(* Logix 5000 project; controller Transcat_L33ER vendor 1 type 14 code 107 rev 32.11; software revision 32.02; part 2 of 2 *)
(* tags used below, declared in another part *)
   alwaysOFF : BOOL;
   AnyAutoRun : BOOL;   // Bit that in on if ANY device is placed into Auto run (to signal pre-start beed)
   AnyManualRun : BOOL;   // Bit that in on if ANY device is placed into manual run (to signal pre-start beed)
   BeaconBlueLight : ALIAS FOR TC_Remote_IO:3:O.3;   // Blue Beacon Light
   BeaconGreenLight : ALIAS FOR TC_Remote_IO:3:O.2;   // Green Beacon Light
   BeaconRedLight : ALIAS FOR TC_Remote_IO:3:O.0;   // Red Beacon Light
   BeaconYellowLight : ALIAS FOR TC_Remote_IO:3:O.1;   // Yellow Beacon Light
   Beep : BOOL;   // Bit to Activte Beacon Alarm
   BeepNew : ALIAS FOR TC_Remote_IO:3:O.4;
   Device : Device[20];
   FT103 : BronkhorstFlowMeter;
   FT104 : BronkhorstFlowMeter;
   FT105 : BronkhorstFlowMeter;
   GF101 : Thayer_WB_Feeder;   // Thayer 1 Tags
   GF201 : Thayer_WB_Feeder;   // Thayer 2 Tags
   GF301 : Acrison_Feeder;   // GF103 - Small Feeder 1
   GreenFlashingOff : TIMER;
   GreenFlashingOn : TIMER;
   HMI_AllReset : BOOL;   // Bit to reset Auto/Man, AutoRun, RecipeRun, TimedRunEnable to 0 from HMI
   MSG_FROM_SLC500 : INT[10];
   MX101 : Howes_Mixer;
   MX201 : Howes_Mixer;
   StartBeepTimer : TIMER;   // Timer to sound the beep alarm before starting a device
   UpperHowesSpeed : INT;
   VF101 : Acrison_Feeder;   // Medium Feeder Tags
   VF201 : Acrison_Feeder;   // Small Feeder 2 Tags
   YellowFlashOff : TIMER;
   YellowFlashOn : TIMER;
   ZS101_RPM_Speed_UpperHowes : ALIAS FOR TC_Remote_IO:1:I.Ch3Data;   // Upper Howes Zero Speed Sensor RPM
   ZS102_RPM_Speed_LowerHowes : ALIAS FOR TC_Remote_IO:1:I.Ch4Data;   // Lower Howes Zero Speed Sensor RPM
(* MainProgram, continued *)

ROUTINE Light_Beacon   (* ladder *)
// Indicator Light Beacon
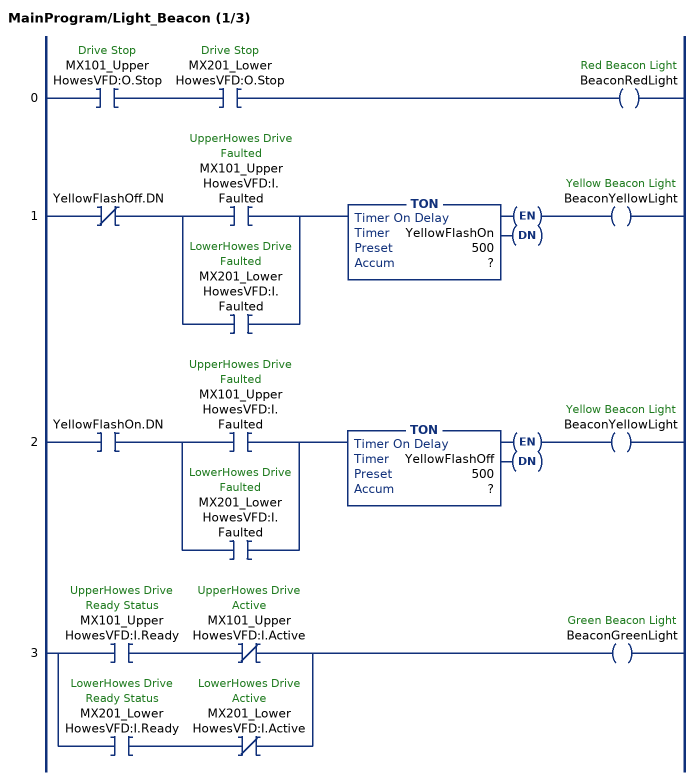
   0: XIC(MX101_UpperHowesVFD:O.Stop)XIC(MX201_LowerHowesVFD:O.Stop)OTE(BeaconRedLight);
   1: XIO(YellowFlashOff.DN)[XIC(MX101_UpperHowesVFD:I.Faulted) ,XIC(MX201_LowerHowesVFD:I.Faulted) ]TON(YellowFlashOn,?,?)OTE(BeaconYellowLight);
   2: XIC(YellowFlashOn.DN)[XIC(MX101_UpperHowesVFD:I.Faulted) ,XIC(MX201_LowerHowesVFD:I.Faulted) ]TON(YellowFlashOff,?,?)OTE(BeaconYellowLight);
   3: [XIC(MX101_UpperHowesVFD:I.Ready) XIO(MX101_UpperHowesVFD:I.Active) ,XIC(MX201_LowerHowesVFD:I.Ready) XIO(MX201_LowerHowesVFD:I.Active) ]OTE(BeaconGreenLight);
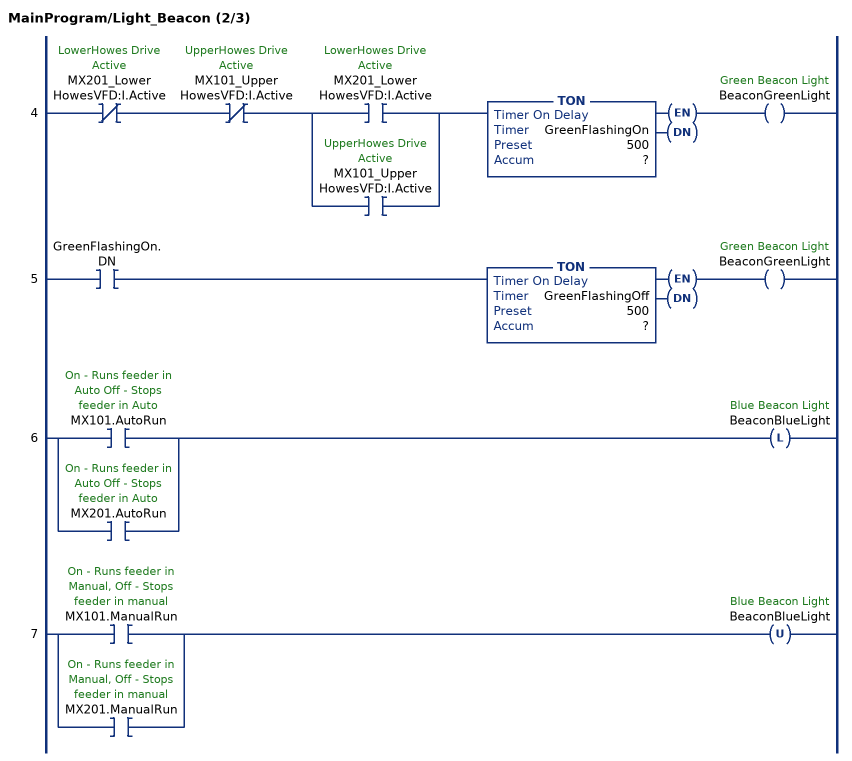
   4: XIO(MX201_LowerHowesVFD:I.Active)XIO(MX101_UpperHowesVFD:I.Active)[XIC(MX201_LowerHowesVFD:I.Active) ,XIC(MX101_UpperHowesVFD:I.Active) ]TON(GreenFlashingOn,?,?)OTE(BeaconGreenLight);
   5: XIC(GreenFlashingOn.DN)TON(GreenFlashingOff,?,?)OTE(BeaconGreenLight);
   6: [XIC(MX101.AutoRun) ,XIC(MX201.AutoRun) ]OTL(BeaconBlueLight);
   7: [XIC(MX101.ManualRun) ,XIC(MX201.ManualRun) ]OTU(BeaconBlueLight);
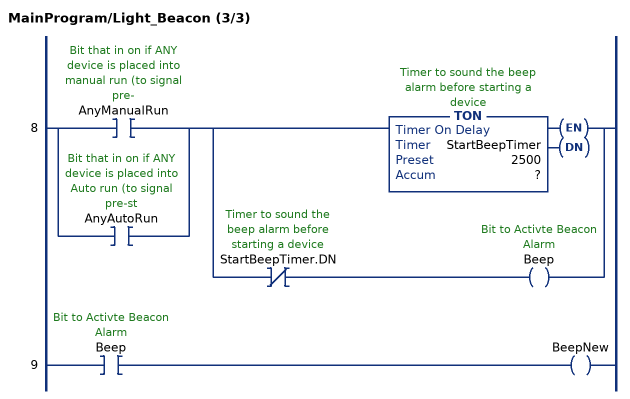
   8: [XIC(AnyManualRun) ,XIC(AnyAutoRun) ][TON(StartBeepTimer,?,?) ,XIO(StartBeepTimer.DN) OTE(Beep) ];
   9: XIC(Beep)OTE(BeepNew);
END_ROUTINE

ROUTINE MainRoutine   (* ladder *)
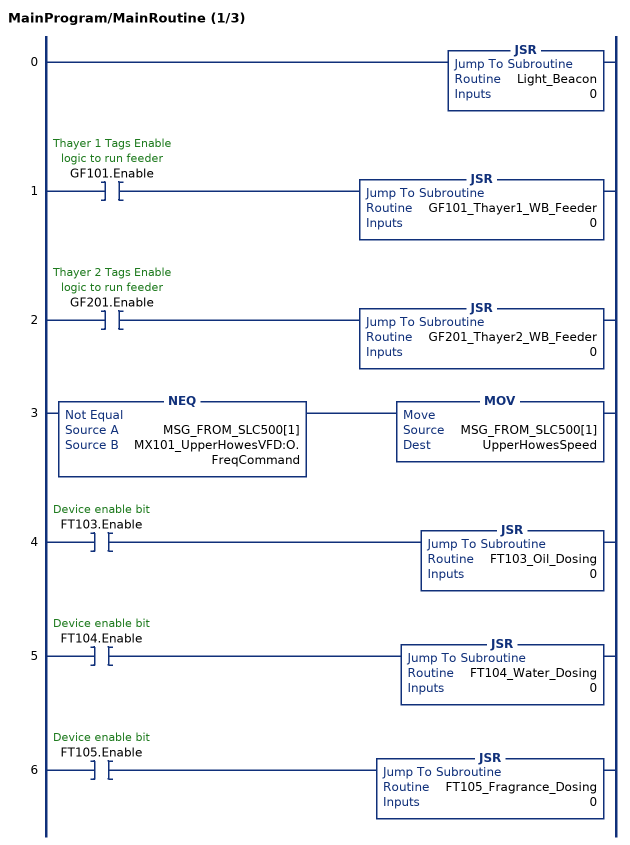
   0: JSR(Light_Beacon,0);
   1: XIC(GF101.Enable)JSR(GF101_Thayer1_WB_Feeder,0);
   2: XIC(GF201.Enable)JSR(GF201_Thayer2_WB_Feeder,0);
   3: NEQ(MSG_FROM_SLC500[1],MX101_UpperHowesVFD:O.FreqCommand)MOV(MSG_FROM_SLC500[1],UpperHowesSpeed);
   4: XIC(FT103.Enable)JSR(FT103_Oil_Dosing,0);
   5: XIC(FT104.Enable)JSR(FT104_Water_Dosing,0);
   6: XIC(FT105.Enable)JSR(FT105_Fragrance_Dosing,0);
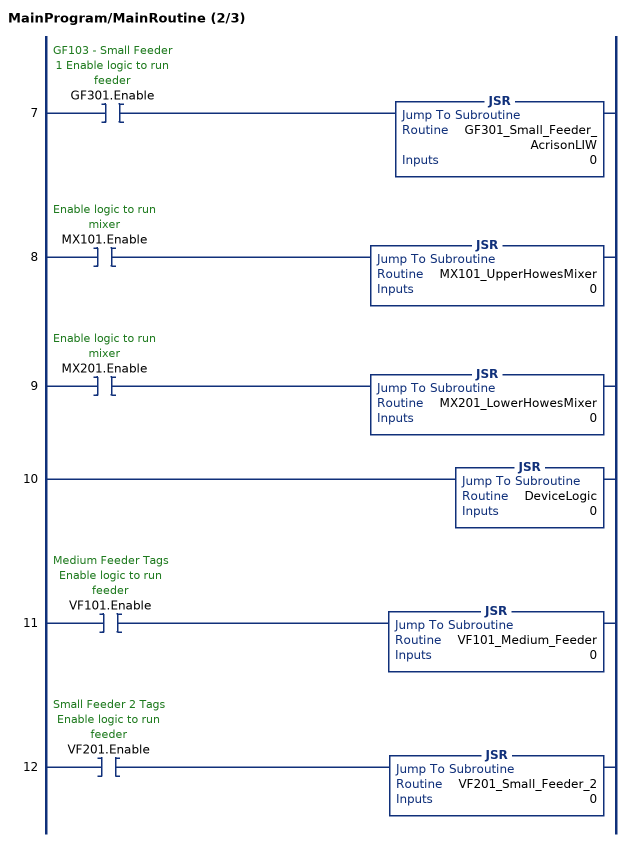
   7: XIC(GF301.Enable)JSR(GF301_Small_Feeder_AcrisonLIW,0);
   8: XIC(MX101.Enable)JSR(MX101_UpperHowesMixer,0);
   9: XIC(MX201.Enable)JSR(MX201_LowerHowesMixer,0);
   10: JSR(DeviceLogic,0);
   11: XIC(VF101.Enable)JSR(VF101_Medium_Feeder,0);
   12: XIC(VF201.Enable)JSR(VF201_Small_Feeder_2,0);
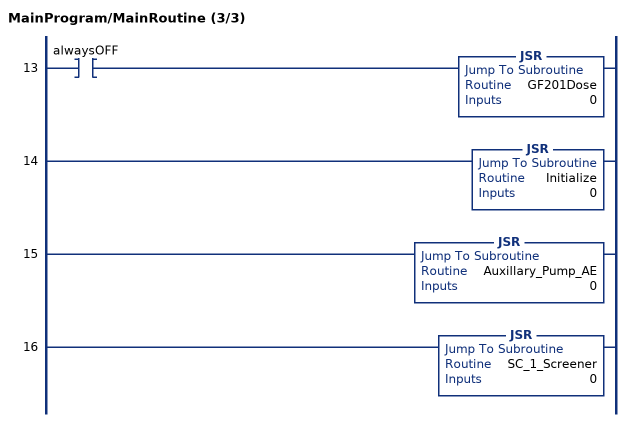
   13: XIC(alwaysOFF)JSR(GF201Dose,0);
   14: JSR(Initialize,0);
   15: JSR(Auxillary_Pump_AE,0);
   16: JSR(SC_1_Screener,0);
END_ROUTINE

ROUTINE MX101_UpperHowesMixer   (* ladder *)
// Upper Howes Mixer Specific (non Iteration) Control Logic
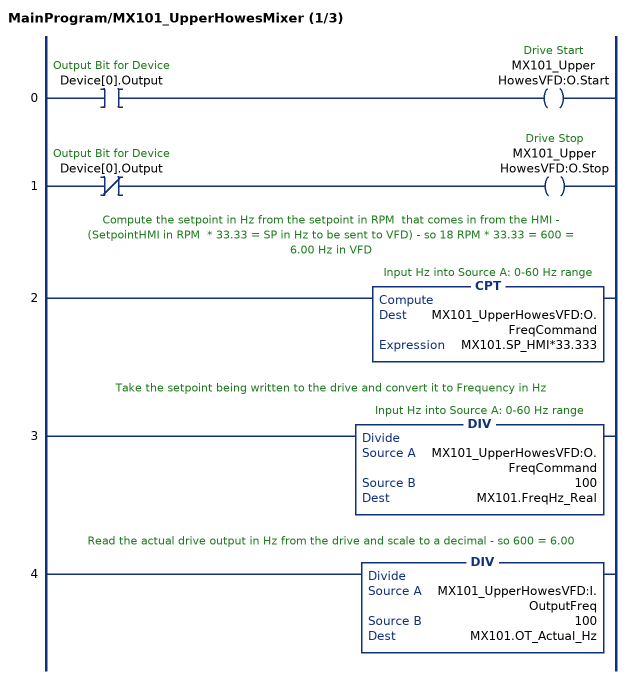
   0: XIC(Device[0].Output)OTE(MX101_UpperHowesVFD:O.Start);
   1: XIO(Device[0].Output)OTE(MX101_UpperHowesVFD:O.Stop);
   // Compute the setpoint in Hz from the setpoint in RPM  that comes in from the HMI - (SetpointHMI in RPM  * 33.33 = SP in Hz to be sent to VFD) - so 18 RPM * 33.33 = 600 = 6.00 Hz in VFD
   2: CPT(MX101_UpperHowesVFD:O.FreqCommand,MX101.SP_HMI*33.333);
   // Take the setpoint being written to the drive and convert it to Frequency in Hz
   3: DIV(MX101_UpperHowesVFD:O.FreqCommand,100,MX101.FreqHz_Real);
   // Read the actual drive output in Hz from the drive and scale to a decimal - so 600 = 6.00
   4: DIV(MX101_UpperHowesVFD:I.OutputFreq,100,MX101.OT_Actual_Hz);
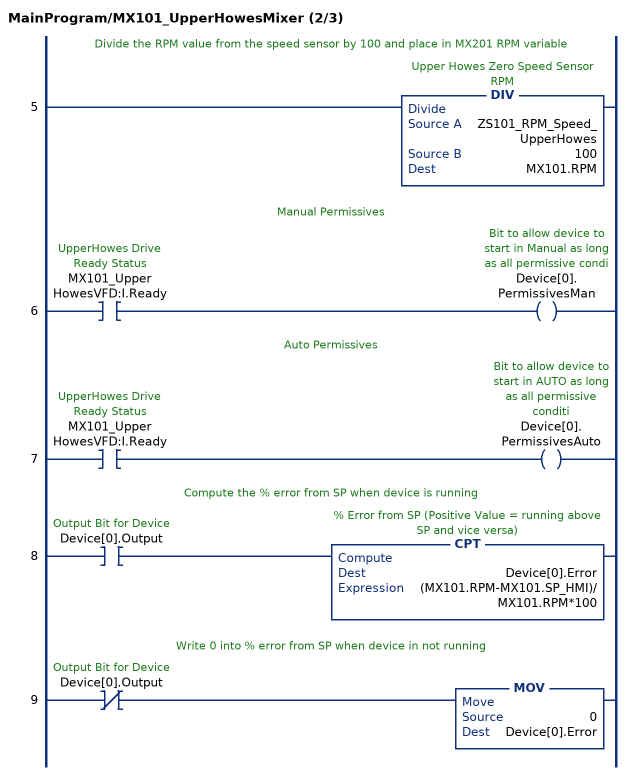
   // Divide the RPM value from the speed sensor by 100 and place in MX201 RPM variable
   5: DIV(ZS101_RPM_Speed_UpperHowes,100,MX101.RPM);
   // Manual Permissives
   6: XIC(MX101_UpperHowesVFD:I.Ready)OTE(Device[0].PermissivesMan);
   // Auto Permissives
   7: XIC(MX101_UpperHowesVFD:I.Ready)OTE(Device[0].PermissivesAuto);
   // Compute the % error from SP when device is running
   8: XIC(Device[0].Output)CPT(Device[0].Error,(MX101.RPM-MX101.SP_HMI)/MX101.RPM*100);
   // Write 0 into % error from SP when device in not running
   9: XIO(Device[0].Output)MOV(0,Device[0].Error);
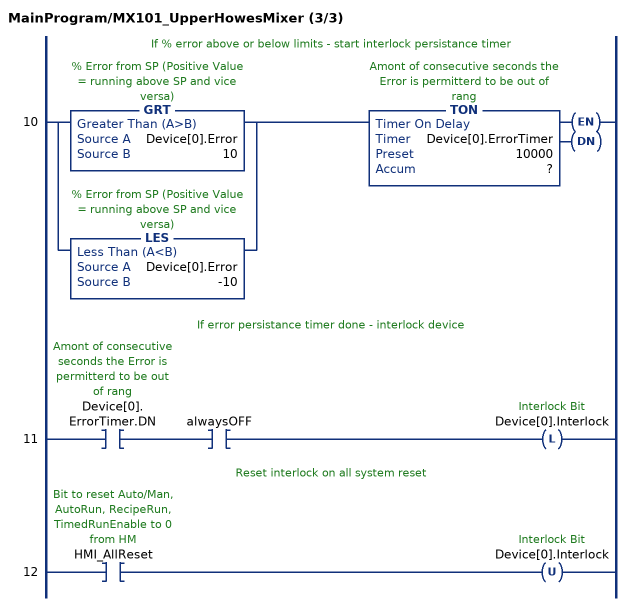
   // If % error above or below limits - start interlock persistance timer
   10: [GRT(Device[0].Error,10) ,LES(Device[0].Error,-10) ]TON(Device[0].ErrorTimer,?,?);
   // If error persistance timer done - interlock device
   11: XIC(Device[0].ErrorTimer.DN)XIC(alwaysOFF)OTL(Device[0].Interlock);
   // Reset interlock on all system reset
   12: XIC(HMI_AllReset)OTU(Device[0].Interlock);
END_ROUTINE

ROUTINE MX201_LowerHowesMixer   (* ladder *)
// Lower Howes Mixer Control Logic not associated with Device Iteration Logic
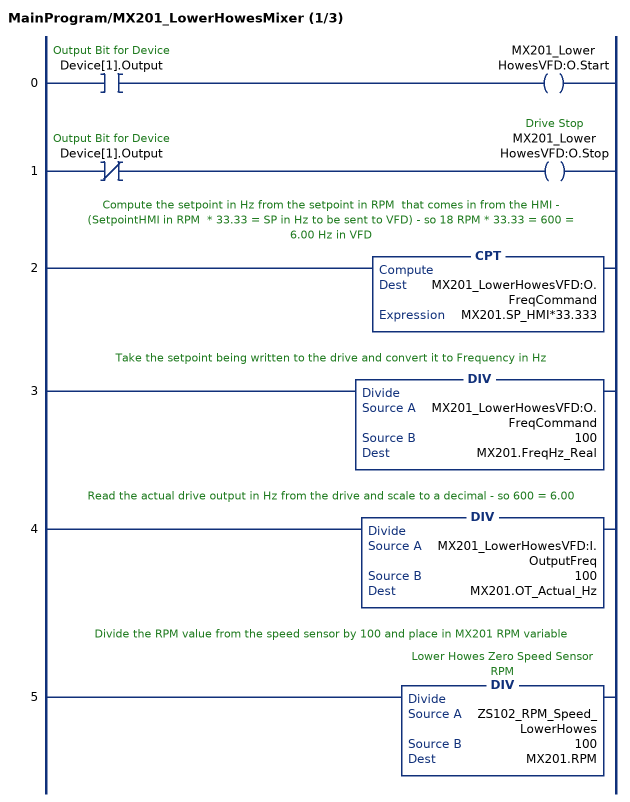
   0: XIC(Device[1].Output)OTE(MX201_LowerHowesVFD:O.Start);
   1: XIO(Device[1].Output)OTE(MX201_LowerHowesVFD:O.Stop);
   // Compute the setpoint in Hz from the setpoint in RPM  that comes in from the HMI - (SetpointHMI in RPM  * 33.33 = SP in Hz to be sent to VFD) - so 18 RPM * 33.33 = 600 = 6.00 Hz in VFD
   2: CPT(MX201_LowerHowesVFD:O.FreqCommand,MX201.SP_HMI*33.333);
   // Take the setpoint being written to the drive and convert it to Frequency in Hz
   3: DIV(MX201_LowerHowesVFD:O.FreqCommand,100,MX201.FreqHz_Real);
   // Read the actual drive output in Hz from the drive and scale to a decimal - so 600 = 6.00
   4: DIV(MX201_LowerHowesVFD:I.OutputFreq,100,MX201.OT_Actual_Hz);
   // Divide the RPM value from the speed sensor by 100 and place in MX201 RPM variable
   5: DIV(ZS102_RPM_Speed_LowerHowes,100,MX201.RPM);
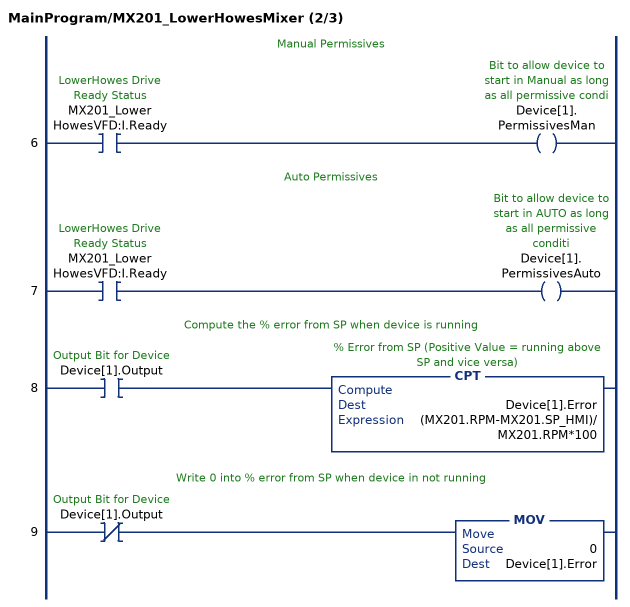
   // Manual Permissives
   6: XIC(MX201_LowerHowesVFD:I.Ready)OTE(Device[1].PermissivesMan);
   // Auto Permissives
   7: XIC(MX201_LowerHowesVFD:I.Ready)OTE(Device[1].PermissivesAuto);
   // Compute the % error from SP when device is running
   8: XIC(Device[1].Output)CPT(Device[1].Error,(MX201.RPM-MX201.SP_HMI)/MX201.RPM*100);
   // Write 0 into % error from SP when device in not running
   9: XIO(Device[1].Output)MOV(0,Device[1].Error);
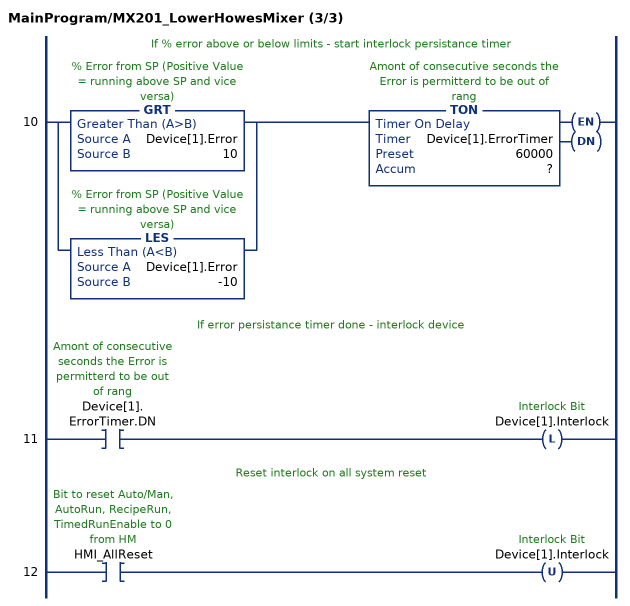
   // If % error above or below limits - start interlock persistance timer
   10: [GRT(Device[1].Error,10) ,LES(Device[1].Error,-10) ]TON(Device[1].ErrorTimer,?,?);
   // If error persistance timer done - interlock device
   11: XIC(Device[1].ErrorTimer.DN)OTL(Device[1].Interlock);
   // Reset interlock on all system reset
   12: XIC(HMI_AllReset)OTU(Device[1].Interlock);
END_ROUTINE

ROUTINE SC_1_Screener   (* ladder *)
// Screener
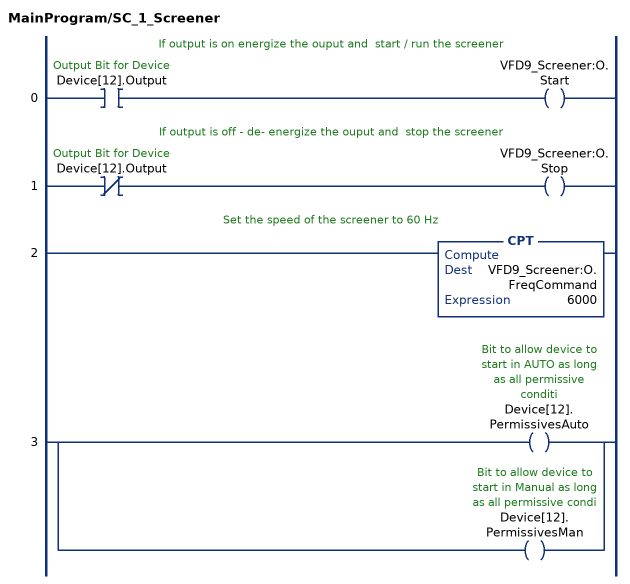
   // If output is on energize the ouput and  start / run the screener
   0: XIC(Device[12].Output)OTE(VFD9_Screener:O.Start);
   // If output is off - de- energize the ouput and  stop the screener
   1: XIO(Device[12].Output)OTE(VFD9_Screener:O.Stop);
   // Set the speed of the screener to 60 Hz
   2: CPT(VFD9_Screener:O.FreqCommand,6000);
   3: [OTE(Device[12].PermissivesAuto) ,OTE(Device[12].PermissivesMan) ];
END_ROUTINE

ROUTINE VF101_Medium_Feeder   (* ladder *)
// Control Logix Specific to VF101 Medium Feeder
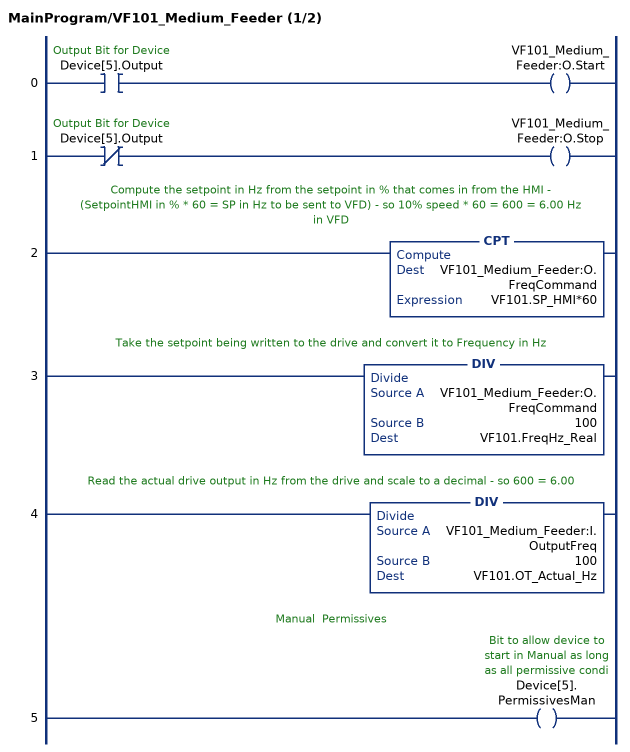
   0: XIC(Device[5].Output)OTE(VF101_Medium_Feeder:O.Start);
   1: XIO(Device[5].Output)OTE(VF101_Medium_Feeder:O.Stop);
   // Compute the setpoint in Hz from the setpoint in % that comes in from the HMI - (SetpointHMI in % * 60 = SP in Hz to be sent to VFD) - so 10% speed * 60 = 600 = 6.00 Hz in VFD
   2: CPT(VF101_Medium_Feeder:O.FreqCommand,VF101.SP_HMI*60);
   // Take the setpoint being written to the drive and convert it to Frequency in Hz
   3: DIV(VF101_Medium_Feeder:O.FreqCommand,100,VF101.FreqHz_Real);
   // Read the actual drive output in Hz from the drive and scale to a decimal - so 600 = 6.00
   4: DIV(VF101_Medium_Feeder:I.OutputFreq,100,VF101.OT_Actual_Hz);
   // Manual  Permissives
   5: OTE(Device[5].PermissivesMan);
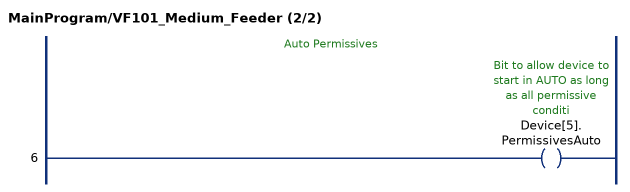
   // Auto Permissives
   6: OTE(Device[5].PermissivesAuto);
END_ROUTINE

ROUTINE VF201_Small_Feeder_2   (* ladder *)
// Acison Small Feeder Control
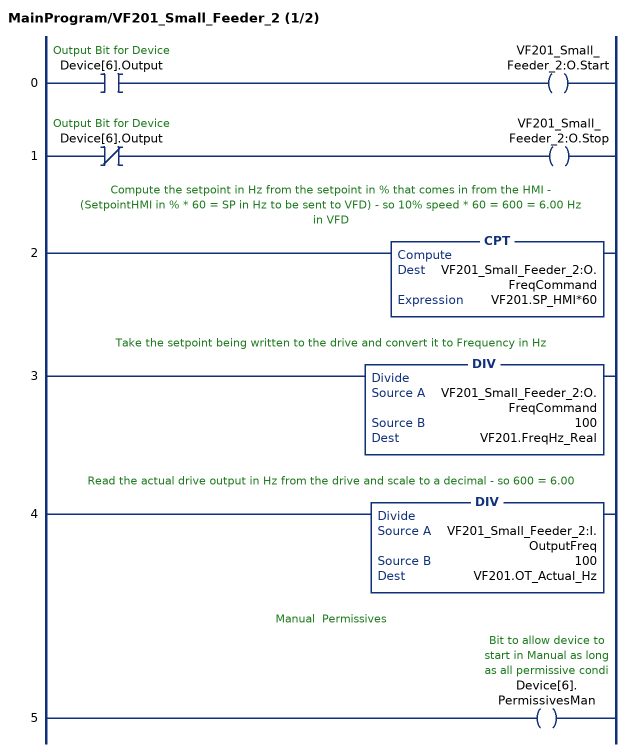
   0: XIC(Device[6].Output)OTE(VF201_Small_Feeder_2:O.Start);
   1: XIO(Device[6].Output)OTE(VF201_Small_Feeder_2:O.Stop);
   // Compute the setpoint in Hz from the setpoint in % that comes in from the HMI - (SetpointHMI in % * 60 = SP in Hz to be sent to VFD) - so 10% speed * 60 = 600 = 6.00 Hz in VFD
   2: CPT(VF201_Small_Feeder_2:O.FreqCommand,VF201.SP_HMI*60);
   // Take the setpoint being written to the drive and convert it to Frequency in Hz
   3: DIV(VF201_Small_Feeder_2:O.FreqCommand,100,VF201.FreqHz_Real);
   // Read the actual drive output in Hz from the drive and scale to a decimal - so 600 = 6.00
   4: DIV(VF201_Small_Feeder_2:I.OutputFreq,100,VF201.OT_Actual_Hz);
   // Manual  Permissives
   5: OTE(Device[6].PermissivesMan);
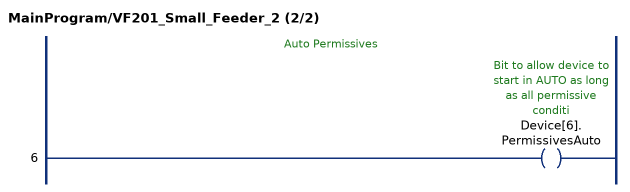
   // Auto Permissives
   6: OTE(Device[6].PermissivesAuto);
END_ROUTINE
END_PROGRAM
